FUNCTION_BLOCK F_NOT_BOOL (* standard boolean NOT function *)
  (* Standard: 61131-3; Classification: standard boolean function; Description: Copyright (c) 2011 TU Wien ACIN This program and the accompanying materials are made available under the terms of the Eclipse Public License 2.0 which is available at https://www.eclipse.org/legal/epl-2.0/ SPDX-License-Identifier: EPL-2.0 *)
  (* Version 1.0, 2011-06-21, Monika Wenger, TU Wien ACIN, initial API and implementation and/or initial documentation *)
  (* Version 3.0, 2025-04-14, Patrick Aigner, changed package *)
  PACKAGE iec61131::bitwiseOperators;
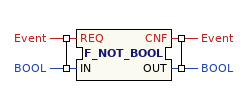
  EVENT_INPUT
    REQ WITH IN; (* Service Request *)
  END_EVENT
  EVENT_OUTPUT
    CNF WITH OUT; (* Confirmation of Requested Service *)
  END_EVENT
  VAR_INPUT
    IN : BOOL; (* Input *)
  END_VAR
  VAR_OUTPUT
    OUT : BOOL; (* Output *)
  END_VAR
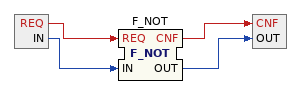
  FBS
    F_NOT : iec61131::bitwiseOperators::F_NOT;
  END_FBS
  EVENT_CONNECTIONS
    REQ TO F_NOT.REQ;
    F_NOT.CNF TO CNF;
  END_CONNECTIONS
  DATA_CONNECTIONS
    IN TO F_NOT.IN;
    F_NOT.OUT TO OUT;
  END_CONNECTIONS
END_FUNCTION_BLOCK
